PROGRAM MAIN
VAR
	test:FB_GaugeModbus;
	
END_VAR

test(IP:='172.21.84.44',nMBAddr:=2048(*8#4000*),iBitOffset:=24);

END_PROGRAM

(* stored: Version 1.1.0.1, ProductVersion 3.1.4022.18
   POU MAIN: Id {7bbf0460-3de1-4d39-9a4c-ffbbff143741}, SpecialFunc None *)
